{attribute 'qualified_only'}
{attribute 'strict'}
TYPE E_Number :
(
	Init    := -32768,
	Start 	:= 0,
	Done	:= 32767
)INT;
END_TYPE

(* stored: Version 1.1.0.1
   DUT E_Number: Id {6c594fbe-a1d3-4b2d-af82-ae3ef2090850} *)
